// TIA Portal V19 export
TYPE "IF Burkett Type 8691 IO"
   STRUCT
      StandardStructure : Struct
         Header : Struct
            NumberParameter : Int := 56;   // Number of device parameters (Device Identification + Device Parameter)
            AdressParamDownLoad : Int := 20;   // Start adress for ParamDownload signals in this struct
            AdressDeviceIndent : Int := 44;   // Start adress for Device Identification Parameters in this struct
            AdressApplicSpez : Int := 700;   // Start adress ApplicationSpezificTag
            AdressDeviceParam : Int := 1110;   // Start adress for Device Parameters in this Area
            AdressKommando : Int := 1970;   // Start adress for Device Commandos
            NumberCommandos : Int := 4;   // Number of Commandos of the device
            Spare01 : Int;   // spare
            Spare02 : Int;   // spare
            Spare03 : Int;   // spare
         END_STRUCT;
         Paramdownload : Struct
            ParamDownLoadStart : Struct   // Parameter Download Start (Only if master and device are V1.1)
               BlockStat : DWord;   // function block status
               IOLStat : DWord;   // IO-Link Status
            END_STRUCT;
            ParamDownLoadEnd : Struct   // Parameter Download End (Only if master and device are V1.1)
               BlockStat : DWord;   // function block status
               IOLStat : DWord;   // IO-Link Status
            END_STRUCT;
            ParamDownLoadStore : Struct   // Parameter Download Store (Only if master and device are V1.1)
               BlockStat : DWord;   // function block status
               IOLStat : DWord;   // IO-Link Status
            END_STRUCT;
         END_STRUCT;
         DeviceIndentification : Struct   // device indentification parameter
            V_VendorName : Struct   // Vendor Name
               Text : String[64];
               Index : Int := 16;   // parameter index
               Subindex : Int;   // parameter subindex
               Length : Int := 64;   // parameter length in BYTE for writing
               BlockStat : DWord;   // function block status
               IOLStat : DWord;   // IO-Link Status
               RelRead : Bool := TRUE;   // reading release
               RelWrite : Bool;   // writing release
            END_STRUCT;
            V_VendorText : Struct   // Vendor Text
               Text : String[64];
               Index : Int := 17;   // parameter index
               Subindex : Int;   // parameter subindex
               Length : Int := 64;   // parameter length in BYTE for writing
               BlockStat : DWord;   // function block status
               IOLStat : DWord;   // IO-Link Status
               RelRead : Bool := TRUE;   // reading release
               RelWrite : Bool;   // writing release
            END_STRUCT;
            V_ProductName : Struct   // Product Name
               Text : String[64];
               Index : Int := 18;   // parameter index
               Subindex : Int;   // parameter subindex
               Length : Int := 64;   // parameter length in BYTE for writing
               BlockStat : DWord;   // function block status
               IOLStat : DWord;   // IO-Link Status
               RelRead : Bool := TRUE;   // reading release
               RelWrite : Bool;   // writing release
            END_STRUCT;
            V_ProductID : Struct   // Product ID
               Text : String[64];
               Index : Int := 19;   // parameter index
               Subindex : Int;   // parameter subindex
               Length : Int := 64;   // parameter length in BYTE for writing
               BlockStat : DWord;   // function block status
               IOLStat : DWord;   // IO-Link Status
               RelRead : Bool := TRUE;   // reading release
               RelWrite : Bool;   // writing release
            END_STRUCT;
            V_ProductText : Struct   // Product Text
               Text : String[64];
               Index : Int := 20;   // parameter index
               Subindex : Int;   // parameter subindex
               Length : Int := 64;   // parameter length in BYTE for writing
               BlockStat : DWord;   // function block status
               IOLStat : DWord;   // IO-Link Status
               RelRead : Bool := TRUE;   // reading release
               RelWrite : Bool;   // writing release
            END_STRUCT;
            V_SerialNumber : Struct   // Serial Number
               Text : String[64];
               Index : Int := 21;   // parameter index
               Subindex : Int;   // parameter subindex
               Length : Int := 16;   // parameter length in BYTE for writing
               BlockStat : DWord;   // function block status
               IOLStat : DWord;   // IO-Link Status
               RelRead : Bool := TRUE;   // reading release
               RelWrite : Bool;   // writing release
            END_STRUCT;
            V_HardwareRevision : Struct   // Hardware Version
               Text : String[64];
               Index : Int := 22;   // parameter index
               Subindex : Int;   // parameter subindex
               Length : Int := 64;   // parameter length in BYTE for writing
               BlockStat : DWord;   // function block status
               IOLStat : DWord;   // IO-Link Status
               RelRead : Bool := TRUE;   // reading release
               RelWrite : Bool;   // writing release
            END_STRUCT;
            V_FirmwareRevision : Struct   // Firmware Version
               Text : String[64];
               Index : Int := 23;   // parameter index
               Subindex : Int;   // parameter subindex
               Length : Int := 64;   // parameter length in BYTE for writing
               BlockStat : DWord;   // function block status
               IOLStat : DWord;   // IO-Link Status
               RelRead : Bool := TRUE;   // reading release
               RelWrite : Bool;   // writing release
            END_STRUCT;
         END_STRUCT;
         ApplicationSpecificTag : Struct   // AppliciationSpecificTag
            V_ApplicationSpecificTa : Struct   // Application Specific Tag
               Text : String[64];
               Index : Int := 24;   // parameter index
               Subindex : Int;   // parameter subindex
               Length : Int := 19;   // parameter length in BYTE for writing
               BlockStat : DWord;   // function block status
               IOLStat : DWord;   // IO-Link Status
               RelRead : Bool := TRUE;   // reading release
               RelWrite : Bool := TRUE;   // writing release
            END_STRUCT;
            V_UniqueDeviceName : Struct   // Name of Device
               Text : String[64];
               Index : Int := 8194;   // parameter index
               Subindex : Int := 1;   // parameter subindex
               Length : Int := 19;   // parameter length in BYTE for writing
               BlockStat : DWord;   // function block status
               IOLStat : DWord;   // IO-Link Status
               RelRead : Bool := TRUE;   // reading release
               RelWrite : Bool := TRUE;   // writing release
            END_STRUCT;
            V_LocationInformation : Struct   // Information about device location
               Text : String[64];
               Index : Int := 8194;   // parameter index
               Subindex : Int := 2;   // parameter subindex
               Length : Int := 19;   // parameter length in BYTE for writing
               BlockStat : DWord;   // function block status
               IOLStat : DWord;   // IO-Link Status
               RelRead : Bool := TRUE;   // reading release
               RelWrite : Bool := TRUE;   // writing release
            END_STRUCT;
            V_UserDescription : Struct   // Information about device
               Text : String[64];
               Index : Int := 8194;   // parameter index
               Subindex : Int := 3;   // parameter subindex
               Length : Int := 19;   // parameter length in BYTE for writing
               BlockStat : DWord;   // function block status
               IOLStat : DWord;   // IO-Link Status
               RelRead : Bool := TRUE;   // reading release
               RelWrite : Bool := TRUE;   // writing release
            END_STRUCT;
            V_DisplayedDeviceName : Struct   // Device (Tag) name
               Text : String[64];
               Index : Int := 8194;   // parameter index
               Subindex : Int := 4;   // parameter subindex
               Length : Int := 19;   // parameter length in BYTE for writing
               BlockStat : DWord;   // function block status
               IOLStat : DWord;   // IO-Link Status
               RelRead : Bool := TRUE;   // reading release
               RelWrite : Bool := TRUE;   // writing release
            END_STRUCT;
         END_STRUCT;
         DeviceParameters : Struct   // Device Parameters
            Parameter_00 : Struct
               Value : Struct   // Device Status
                  DeviceStatus : Byte;
                  byte_02 : Byte;
                  byte_03 : Byte;
                  byte_04 : Byte;
               END_STRUCT;
               Index : Int := 36;   // parameter index
               Subindex : Int;   // parameter subindex
               Length : Int := 1;   // parameter length in BYTE for writing
               BlockStat : DWord;   // function block status
               IOLStat : DWord;   // IO-Link Status
               RelRead : Bool := TRUE;   // reading release
               RelWrite : Bool;   // writing release
            END_STRUCT;
            Parameter_01 : Struct   // *** Control Head Settings - Index = 11276 ***
               Value : Struct   // Upper (open) tolerance band in mm
                  UTB : Real := 1.5;   // mm
               END_STRUCT;
               Index : Int := 11275;   // parameter index
               Subindex : Int := 1;   // parameter subindex
               Length : Int := 4;   // parameter length in BYTE for writing
               BlockStat : DWord;   // function block status
               IOLStat : DWord;   // IO-Link Status
               RelRead : Bool := TRUE;   // reading release
               RelWrite : Bool := TRUE;   // writing release
            END_STRUCT;
            Parameter_02 : Struct   // Control Head Settings - Lower (closed) tolerance band in mm
               Value : Struct   // Lower (closed) tolerance band in mm
                  LTB : Real := 1.5;   // mm Index = 11276
               END_STRUCT;
               Index : Int := 11275;   // parameter index
               Subindex : Int := 2;   // parameter subindex
               Length : Int := 4;   // parameter length in BYTE for writing
               BlockStat : DWord;   // function block status
               IOLStat : DWord;   // IO-Link Status
               RelRead : Bool := TRUE;   // reading release
               RelWrite : Bool := TRUE;   // writing release
            END_STRUCT;
            Parameter_03 : Struct   // Invert CMD Setpoint value
               Value : Struct   // Parameter Value (must be always 4 Byte)
                  InvertCMD_SP : Byte;   // 0=inversion inactive, 1=inversion inactive
                  Byte01 : Byte;
                  Byte02 : Byte;
                  Byte03 : Byte;
               END_STRUCT;
               Index : Int := 11275;   // parameter index
               Subindex : Int := 3;   // parameter subindex
               Length : Int := 1;   // parameter length in BYTE for writing
               BlockStat : DWord;   // function block status
               IOLStat : DWord;   // IO-Link Status
               RelRead : Bool := TRUE;   // reading release
               RelWrite : Bool := TRUE;   // writing release
            END_STRUCT;
            Parameter_04 : Struct   // Opening Time (CMD)
               Value : Struct   // Parameter Value (must be always 4 Byte)
                  OpeningTime : Int;   // ms
                  Byte02 : Byte;
                  Byte03 : Byte;
               END_STRUCT;
               Index : Int := 11275;   // parameter index
               Subindex : Int := 4;   // parameter subindex
               Length : Int := 2;   // parameter length in BYTE for writing
               BlockStat : DWord;   // function block status
               IOLStat : DWord;   // IO-Link Status
               RelRead : Bool := TRUE;   // reading release
               RelWrite : Bool;   // writing release
            END_STRUCT;
            Parameter_05 : Struct   // Closing Time (CMD)
               Value : Struct   // Parameter Value (must be always 4 Byte)
                  ClosingTime : Int;   // ms
                  Byte02 : Byte;
                  Byte03 : Byte;
               END_STRUCT;
               Index : Int := 11275;   // parameter index
               Subindex : Int := 5;   // parameter subindex
               Length : Int := 2;   // parameter length in BYTE for writing
               BlockStat : DWord;   // function block status
               IOLStat : DWord;   // IO-Link Status
               RelRead : Bool := TRUE;   // reading release
               RelWrite : Bool;   // writing release
            END_STRUCT;
            Parameter_06 : Struct   // Select reaction inevent of setpoint error
               Value : Struct   // Bus error or invalid process data
                  SetpointError : Byte;   // 0=Maintain position, 1=Safety position (pilot valve off)
                  Byte01 : Byte;
                  Byte02 : Byte;
                  Byte03 : Byte;
               END_STRUCT;
               Index : Int := 11275;   // parameter index
               Subindex : Int := 8;   // parameter subindex
               Length : Int := 1;   // parameter length in BYTE for writing
               BlockStat : DWord;   // function block status
               IOLStat : DWord;   // IO-Link Status
               RelRead : Bool := TRUE;   // reading release
               RelWrite : Bool := TRUE;   // writing release
            END_STRUCT;
            Parameter_07 : Struct   // Acitivate or deacitivate local operation
               Value : Struct   // Button for manula operation inside control head
                  DeviceLock : Byte;   // 0=Button enabled, 1=Button disabled
                  Byte01 : Byte;
                  Byte02 : Byte;
                  Byte03 : Byte;
               END_STRUCT;
               Index : Int := 11275;   // parameter index
               Subindex : Int := 12;   // parameter subindex
               Length : Int := 1;   // parameter length in BYTE for writing
               BlockStat : DWord;   // function block status
               IOLStat : DWord;   // IO-Link Status
               RelRead : Bool := TRUE;   // reading release
               RelWrite : Bool := TRUE;   // writing release
            END_STRUCT;
            Parameter_08 : Struct   // *** Teach Functions Index = 11276 ***
               Value : Struct   // Parameter Value (must be always 4 Byte)
                  UpperEndPosition : Real;
               END_STRUCT;
               Index : Int := 11276;   // parameter index
               Subindex : Int := 1;   // parameter subindex
               Length : Int := 4;   // parameter length in BYTE for writing
               BlockStat : DWord;   // function block status
               IOLStat : DWord;   // IO-Link Status
               RelRead : Bool := TRUE;   // reading release
               RelWrite : Bool;   // writing release
            END_STRUCT;
            Parameter_09 : Struct   // *** Teach Functions Index = 11276 ***
               Value : Struct   // Parameter Value (must be always 4 Byte)
                  LowerEndPosition : Real;
               END_STRUCT;
               Index : Int := 11276;   // parameter index
               Subindex : Int := 2;   // parameter subindex
               Length : Int := 4;   // parameter length in BYTE for writing
               BlockStat : DWord;   // function block status
               IOLStat : DWord;   // IO-Link Status
               RelRead : Bool := TRUE;   // reading release
               RelWrite : Bool;   // writing release
            END_STRUCT;
            Parameter_10 : Struct   // *** Teach Functions Index = 11276 ***
               Value : Struct   // Opening Time between tolerance bands
                  Opening_Time : Int;   // ms
                  Byte02 : Byte;
                  Byte03 : Byte;
               END_STRUCT;
               Index : Int := 11276;   // parameter index
               Subindex : Int := 3;   // parameter subindex
               Length : Int := 2;   // parameter length in BYTE for writing
               BlockStat : DWord;   // function block status
               IOLStat : DWord;   // IO-Link Status
               RelRead : Bool := TRUE;   // reading release
               RelWrite : Bool;   // writing release
            END_STRUCT;
            Parameter_11 : Struct   // *** Teach Functions Index = 11276 ***
               Value : Struct   // Closing Time between tolerance bands
                  Closing_Time : Int;   // ms
                  Byte02 : Byte;
                  Byte03 : Byte;
               END_STRUCT;
               Index : Int := 11276;   // parameter index
               Subindex : Int := 4;   // parameter subindex
               Length : Int := 2;   // parameter length in BYTE for writing
               BlockStat : DWord;   // function block status
               IOLStat : DWord;   // IO-Link Status
               RelRead : Bool := TRUE;   // reading release
               RelWrite : Bool;   // writing release
            END_STRUCT;
            Parameter_12 : Struct   // *** Teach Functions Index = 11276 ***
               Value : Struct   // Parameter Value (must be always 4 Byte)
                  Stroke : Real;   // Valve stroke in mm
               END_STRUCT;
               Index : Int := 11276;   // parameter index
               Subindex : Int := 5;   // parameter subindex
               Length : Int := 4;   // parameter length in BYTE for writing
               BlockStat : DWord;   // function block status
               IOLStat : DWord;   // IO-Link Status
               RelRead : Bool := TRUE;   // reading release
               RelWrite : Bool;   // writing release
            END_STRUCT;
            Parameter_14 : Struct   // Is Teached
               Value : Struct   // Indicates successful completion of a teach funtion
                  IsTeached : Byte;   // 0=Device has not been taught, 1=Device taught
                  Byte01 : Byte;
                  Byte02 : Byte;
                  Byte03 : Byte;
               END_STRUCT;
               Index : Int := 11276;   // parameter index
               Subindex : Int := 6;   // parameter subindex
               Length : Int := 1;   // parameter length in BYTE for writing
               BlockStat : DWord;   // function block status
               IOLStat : DWord;   // IO-Link Status
               RelRead : Bool := TRUE;   // reading release
               RelWrite : Bool;   // writing release
            END_STRUCT;
            Parameter_15 : Struct   // Teach function State
               Value : Struct   // 0=complete,1=Initialisation,2=End Position1,3=End Position2,4=Check Stroke,
                  TeachFuncState : Byte;   // 5=DetermineSwitchingTime,-1=TimeoutEndPos1,-2=TimeoutEndPos2
                  Byte01 : Byte;   // -3=StrokeTooSmall,-4=ErrorDeterminingSwitchingTime,
                  Byte02 : Byte;   // -5=AbortbySafePos, -6=AbortbyUser
                  Byte03 : Byte;
               END_STRUCT;
               Index : Int := 11276;   // parameter index
               Subindex : Int := 7;   // parameter subindex
               Length : Int := 1;   // parameter length in BYTE for writing
               BlockStat : DWord;   // function block status
               IOLStat : DWord;   // IO-Link Status
               RelRead : Bool := TRUE;   // reading release
               RelWrite : Bool;   // writing release
            END_STRUCT;
            Parameter_16 : Struct   // Start Teach function
               Value : Struct
                  TeachFuncStart : Byte;   // 0 = Finished,1 = StartAutomaticTeach, 2 = StartManualTeach
                  Byte01 : Byte;
                  Byte02 : Byte;
                  Byte03 : Byte;
               END_STRUCT;
               Index : Int := 11276;   // parameter index
               Subindex : Int := 8;   // parameter subindex
               Length : Int := 1;   // parameter length in BYTE for writing
               BlockStat : DWord;   // function block status
               IOLStat : DWord;   // IO-Link Status
               RelRead : Bool := TRUE;   // reading release
               RelWrite : Bool := TRUE;   // writing release
            END_STRUCT;
            Parameter_17 : Struct   // Flag shows pneumatic function
               Value : Struct
                  isNO : Byte;   // 0 = Normally Closed (NC), 1 = Normally Open (NO)
                  Byte01 : Byte;
                  Byte02 : Byte;
                  Byte03 : Byte;
               END_STRUCT;
               Index : Int := 11276;   // parameter index
               Subindex : Int := 9;   // parameter subindex
               Length : Int := 1;   // parameter length in BYTE for writing
               BlockStat : DWord;   // function block status
               IOLStat : DWord;   // IO-Link Status
               RelRead : Bool := TRUE;   // reading release
               RelWrite : Bool;   // writing release
            END_STRUCT;
            Parameter_18 : Struct   // Select CMD set-point value source
               Value : Struct
                  CMD_Source : Byte := BYTE#16#01;   // 1 = IO-Link (Cyclic or via SIO),2 = InternalButton, 3 = ManualSPValue(sub0x4)
                  Byte01 : Byte;
                  Byte02 : Byte;
                  Byte03 : Byte;
               END_STRUCT;
               Index : Int := 11277;   // parameter index
               Subindex : Int := 1;   // parameter subindex
               Length : Int := 1;   // parameter length in BYTE for writing
               BlockStat : DWord;   // function block status
               IOLStat : DWord;   // IO-Link Status
               RelRead : Bool := TRUE;   // reading release
               RelWrite : Bool := TRUE;   // writing release
            END_STRUCT;
            Parameter_19 : Struct   // Manual CMD Set-point
               Value : Struct
                  Manual_CMD_SP : Byte;
                  Byte01 : Byte;
                  Byte02 : Byte;
                  Byte03 : Byte;
               END_STRUCT;
               Index : Int := 11277;   // parameter index
               Subindex : Int := 4;   // parameter subindex
               Length : Int := 1;   // parameter length in BYTE for writing
               BlockStat : DWord;   // function block status
               IOLStat : DWord;   // IO-Link Status
               RelRead : Bool := TRUE;   // reading release
               RelWrite : Bool := TRUE;   // writing release
            END_STRUCT;
            Parameter_20 : Struct   // *** Diagnostics , Index = 11278 ***
               Value : Struct
                  TravelAccumlator : Real;   // Valve stem travel in mm
               END_STRUCT;
               Index : Int := 11278;   // parameter index
               Subindex : Int := 1;   // parameter subindex
               Length : Int := 4;   // parameter length in BYTE for writing
               BlockStat : DWord;   // function block status
               IOLStat : DWord;   // IO-Link Status
               RelRead : Bool := TRUE;   // reading release
               RelWrite : Bool;   // writing release
            END_STRUCT;
            Parameter_21 : Struct   // *** Diagnostics , Index = 11278 ***
               Value : Struct
                  TravelAccResettable : Real;   // Valve stem travel in mm
               END_STRUCT;
               Index : Int := 11278;   // parameter index
               Subindex : Int := 2;   // parameter subindex
               Length : Int := 4;   // parameter length in BYTE for writing
               BlockStat : DWord;   // function block status
               IOLStat : DWord;   // IO-Link Status
               RelRead : Bool := TRUE;   // reading release
               RelWrite : Bool;   // writing release
            END_STRUCT;
            Parameter_22 : Struct   // Travel Accumulator in mm, Activate or deactivate maintenance threshold
               Value : Struct
                  TravelAccLimit : Real;   // Travel Acc Limit in mm
               END_STRUCT;
               Index : Int := 11278;   // parameter index
               Subindex : Int := 3;   // parameter subindex
               Length : Int := 4;   // parameter length in BYTE for writing
               BlockStat : DWord;   // function block status
               IOLStat : DWord;   // IO-Link Status
               RelRead : Bool := TRUE;   // reading release
               RelWrite : Bool := TRUE;   // writing release
            END_STRUCT;
            Parameter_23 : Struct   // Valve Cycles
               Value : Struct
                  ValveCycles : DInt;   // # of Valve Cycles
               END_STRUCT;
               Index : Int := 11278;   // parameter index
               Subindex : Int := 4;   // parameter subindex
               Length : Int := 4;   // parameter length in BYTE for writing
               BlockStat : DWord;   // function block status
               IOLStat : DWord;   // IO-Link Status
               RelRead : Bool := TRUE;   // reading release
               RelWrite : Bool;   // writing release
            END_STRUCT;
            Parameter_24 : Struct   // Valve Cycles Resetable
               Value : Struct
                  ValveCyclesResettable : DInt;   // # of Valve Cycles
               END_STRUCT;
               Index : Int := 11278;   // parameter index
               Subindex : Int := 5;   // parameter subindex
               Length : Int := 4;   // parameter length in BYTE for writing
               BlockStat : DWord;   // function block status
               IOLStat : DWord;   // IO-Link Status
               RelRead : Bool := TRUE;   // reading release
               RelWrite : Bool;   // writing release
            END_STRUCT;
            Parameter_25 : Struct   // Valve Cycles Limit
               Value : Struct   // ValveCyclesResetable > ValveCyclesLimit = Activate Maintenance Warning
                  ValveCyclesLimit : DInt;   // # of Valve Cycles
               END_STRUCT;
               Index : Int := 11278;   // parameter index
               Subindex : Int := 6;   // parameter subindex
               Length : Int := 4;   // parameter length in BYTE for writing
               BlockStat : DWord;   // function block status
               IOLStat : DWord;   // IO-Link Status
               RelRead : Bool := TRUE;   // reading release
               RelWrite : Bool := TRUE;   // writing release
            END_STRUCT;
            Parameter_26 : Struct   // Operating Time Resettable
               Value : Struct   // Sum of time device recieving operating voltage
                  OperateTimeResettable : DInt;   // time in seconds
               END_STRUCT;
               Index : Int := 11278;   // parameter index
               Subindex : Int := 7;   // parameter subindex
               Length : Int := 4;   // parameter length in BYTE for writing
               BlockStat : DWord;   // function block status
               IOLStat : DWord;   // IO-Link Status
               RelRead : Bool := TRUE;   // reading release
               RelWrite : Bool;   // writing release
            END_STRUCT;
            Parameter_27 : Struct   // Operating Time Limit
               Value : Struct   // OperateTimeResetable > OperateTimeLimit = Activate Maintenance Warning
                  OperateTimeLimit : DInt;   // time in seconds
               END_STRUCT;
               Index : Int := 11278;   // parameter index
               Subindex : Int := 8;   // parameter subindex
               Length : Int := 4;   // parameter length in BYTE for writing
               BlockStat : DWord;   // function block status
               IOLStat : DWord;   // IO-Link Status
               RelRead : Bool := TRUE;   // reading release
               RelWrite : Bool := TRUE;   // writing release
            END_STRUCT;
            Parameter_28 : Struct   // Diagnostics Command
               Value : Struct   // Bit0=ResetSwitchingCycles, Bit1=ResetTravelACC, Bit2=ResetOperateTime
                  Diag_CMD : Byte;   // Bit3=Reset#OfOpeningTimeTimeouts,Bit4=Reset#OfClosingTimeTimeouts,
                  Byte01 : Byte;   // Bit5=CopyMeasuredSwitchingTimes, Bit6=ResetNoOfSwitchingTimeTimeouts
                  Byte02 : Byte;
                  Byte03 : Byte;
               END_STRUCT;
               Index : Int := 11278;   // parameter index
               Subindex : Int := 9;   // parameter subindex
               Length : Int := 1;   // parameter length in BYTE for writing
               BlockStat : DWord;   // function block status
               IOLStat : DWord;   // IO-Link Status
               RelRead : Bool := TRUE;   // reading release
               RelWrite : Bool := TRUE;   // writing release
            END_STRUCT;
            Parameter_29 : Struct   // ** Maximum Opening Time in ms **
               Value : Struct
                  OpeningTimeLimit : Int;   // ms
                  Byte02 : Byte;
                  Byte03 : Byte;
               END_STRUCT;
               Index : Int := 11278;   // parameter index
               Subindex : Int := 10;   // parameter subindex
               Length : Int := 2;   // parameter length in BYTE for writing
               BlockStat : DWord;   // function block status
               IOLStat : DWord;   // IO-Link Status
               RelRead : Bool := TRUE;   // reading release
               RelWrite : Bool := TRUE;   // writing release
            END_STRUCT;
            Parameter_30 : Struct   // ** Maximum Closing Time in ms **
               Value : Struct
                  ClosingTimeLimit : Int;   // ms
                  Byte02 : Byte;
                  Byte03 : Byte;
               END_STRUCT;
               Index : Int := 11278;   // parameter index
               Subindex : Int := 11;   // parameter subindex
               Length : Int := 2;   // parameter length in BYTE for writing
               BlockStat : DWord;   // function block status
               IOLStat : DWord;   // IO-Link Status
               RelRead : Bool := TRUE;   // reading release
               RelWrite : Bool := TRUE;   // writing release
            END_STRUCT;
            Parameter_31 : Struct   // Time Tolerance
               Value : Struct
                  TimeTolerance : Byte;   // %
                  Byte01 : Byte;
                  Byte02 : Byte;
                  Byte03 : Byte;
               END_STRUCT;
               Index : Int := 11278;   // parameter index
               Subindex : Int := 12;   // parameter subindex
               Length : Int := 1;   // parameter length in BYTE for writing
               BlockStat : DWord;   // function block status
               IOLStat : DWord;   // IO-Link Status
               RelRead : Bool := TRUE;   // reading release
               RelWrite : Bool := TRUE;   // writing release
            END_STRUCT;
            Parameter_32 : Struct   // Opening Time Errors
               Value : Struct
                  OpeningTimeErrors : DInt;   // # of Opening Time Errors - Resettable
               END_STRUCT;
               Index : Int := 11278;   // parameter index
               Subindex : Int := 13;   // parameter subindex
               Length : Int := 4;   // parameter length in BYTE for writing
               BlockStat : DWord;   // function block status
               IOLStat : DWord;   // IO-Link Status
               RelRead : Bool := TRUE;   // reading release
               RelWrite : Bool;   // writing release
            END_STRUCT;
            Parameter_33 : Struct   // Closing Time Errors
               Value : Struct
                  ClosingTimeErrors : DInt;   // # of Closing Time Errors - Resettable
               END_STRUCT;
               Index : Int := 11278;   // parameter index
               Subindex : Int := 14;   // parameter subindex
               Length : Int := 4;   // parameter length in BYTE for writing
               BlockStat : DWord;   // function block status
               IOLStat : DWord;   // IO-Link Status
               RelRead : Bool := TRUE;   // reading release
               RelWrite : Bool;   // writing release
            END_STRUCT;
            Parameter_34 : Struct   // Teach Function Counter
               Value : Struct
                  TeachFuncCounter : DInt;   // # of Teach Functions Preformed
               END_STRUCT;
               Index : Int := 11278;   // parameter index
               Subindex : Int := 15;   // parameter subindex
               Length : Int := 4;   // parameter length in BYTE for writing
               BlockStat : DWord;   // function block status
               IOLStat : DWord;   // IO-Link Status
               RelRead : Bool := TRUE;   // reading release
               RelWrite : Bool;   // writing release
            END_STRUCT;
            Parameter_35 : Struct   // Pilot Valve Cycles Counter
               Value : Struct
                  PilotValveCycles : DInt;   // # of Pilot Valve Cycles
               END_STRUCT;
               Index : Int := 11278;   // parameter index
               Subindex : Int := 16;   // parameter subindex
               Length : Int := 4;   // parameter length in BYTE for writing
               BlockStat : DWord;   // function block status
               IOLStat : DWord;   // IO-Link Status
               RelRead : Bool := TRUE;   // reading release
               RelWrite : Bool;   // writing release
            END_STRUCT;
            Parameter_36 : Struct   // Number of Switching Timeouts
               Value : Struct
                  SwitchingTimeouts : DInt;   // # of Switching Timeouts
               END_STRUCT;
               Index : Int := 11278;   // parameter index
               Subindex : Int := 18;   // parameter subindex
               Length : Int := 4;   // parameter length in BYTE for writing
               BlockStat : DWord;   // function block status
               IOLStat : DWord;   // IO-Link Status
               RelRead : Bool := TRUE;   // reading release
               RelWrite : Bool;   // writing release
            END_STRUCT;
            Parameter_37 : Struct   // Select type of switching times for diagnostics
               Value : Struct
                  TimeDiagType : Byte;   // 0=Switching Time Based on CMD, 1=Switching Time Based on position
                  Byte01 : Byte;
                  Byte02 : Byte;
                  Byte03 : Byte;
               END_STRUCT;
               Index : Int := 11278;   // parameter index
               Subindex : Int := 21;   // parameter subindex
               Length : Int := 1;   // parameter length in BYTE for writing
               BlockStat : DWord;   // function block status
               IOLStat : DWord;   // IO-Link Status
               RelRead : Bool := TRUE;   // reading release
               RelWrite : Bool := TRUE;   // writing release
            END_STRUCT;
            Parameter_38 : Struct   // Activate or deactivate switching time timeout detection.
               Value : Struct
                  SwitchingTimeoutDetect : Byte := BYTE#16#01;   // 0=Deactivated, 1=Activated
                  Byte01 : Byte;
                  Byte02 : Byte;
                  Byte03 : Byte;
               END_STRUCT;
               Index : Int := 11278;   // parameter index
               Subindex : Int := 23;   // parameter subindex
               Length : Int := 1;   // parameter length in BYTE for writing
               BlockStat : DWord;   // function block status
               IOLStat : DWord;   // IO-Link Status
               RelRead : Bool := TRUE;   // reading release
               RelWrite : Bool := TRUE;   // writing release
            END_STRUCT;
            Parameter_39 : Struct   // Select max time in ms by which the end position should be reached
               Value : Struct
                  SwitchingTimeout : Int := 500;   // ms
                  Byte02 : Byte;
                  Byte03 : Byte;
               END_STRUCT;
               Index : Int := 11278;   // parameter index
               Subindex : Int := 24;   // parameter subindex
               Length : Int := 2;   // parameter length in BYTE for writing
               BlockStat : DWord;   // function block status
               IOLStat : DWord;   // IO-Link Status
               RelRead : Bool := TRUE;   // reading release
               RelWrite : Bool := TRUE;   // writing release
            END_STRUCT;
            Parameter_40 : Struct   // SIO Mode
               Value : Struct   // Pin 2 / Pin 4
                  SIO_Mode : Byte;   // 0=Open/Close, 1=CMD/Close, 2=CMD/Open
                  Byte01 : Byte;   // ** DEVICE MUST BE RESTARTED IF VALUE CHANGED **
                  Byte02 : Byte;
                  Byte03 : Byte;
               END_STRUCT;
               Index : Int := 11279;   // parameter index
               Subindex : Int := 1;   // parameter subindex
               Length : Int := 1;   // parameter length in BYTE for writing
               BlockStat : DWord;   // function block status
               IOLStat : DWord;   // IO-Link Status
               RelRead : Bool := TRUE;   // reading release
               RelWrite : Bool := TRUE;   // writing release
            END_STRUCT;
            Parameter_41 : Struct   // Output Type
               Value : Struct
                  OutputType : Byte;   // 0=PNP, 1=NPN, 2=PP
                  Byte01 : Byte;   // ** DEVICE MUST BE RESTARTED IF VALUE CHANGED **
                  Byte02 : Byte;
                  Byte03 : Byte;
               END_STRUCT;
               Index : Int := 11279;   // parameter index
               Subindex : Int := 1;   // parameter subindex
               Length : Int := 1;   // parameter length in BYTE for writing
               BlockStat : DWord;   // function block status
               IOLStat : DWord;   // IO-Link Status
               RelRead : Bool := TRUE;   // reading release
               RelWrite : Bool := TRUE;   // writing release
            END_STRUCT;
            Parameter_42 : Struct   // Invert Valve Direction
               Value : Struct
                  InvValveDir : Byte;   // 0=UpperPos/Open, 1=UpperPos/Closed
                  Byte01 : Byte;
                  Byte02 : Byte;
                  Byte03 : Byte;
               END_STRUCT;
               Index : Int := 11268;   // parameter index
               Subindex : Int := 1;   // parameter subindex
               Length : Int := 1;   // parameter length in BYTE for writing
               BlockStat : DWord;   // function block status
               IOLStat : DWord;   // IO-Link Status
               RelRead : Bool := TRUE;   // reading release
               RelWrite : Bool := TRUE;   // writing release
            END_STRUCT;
            Parameter_43 : Struct   // CMD Setpoint Control Mode
               Value : Struct
                  CMD_SP_CNTRL_MODE : Byte;
                  Byte01 : Byte;
                  Byte02 : Byte;
                  Byte03 : Byte;
               END_STRUCT;
               Index : Int := 11268;   // parameter index
               Subindex : Int := 2;   // parameter subindex
               Length : Int := 1;   // parameter length in BYTE for writing
               BlockStat : DWord;   // function block status
               IOLStat : DWord;   // IO-Link Status
               RelRead : Bool := TRUE;   // reading release
               RelWrite : Bool := TRUE;   // writing release
            END_STRUCT;
         END_STRUCT;
         Commando : Struct   // Commandos
            Commando_01 : Struct   // Device Reset
               Value : Byte := BYTE#16#80;   // 128
               Index : Int := 2;   // parameter index
               Subindex : Int;   // parameter subindex
               Length : Int := 1;   // parameter length in BYTE for writing
               BlockStat : DWord;   // function block status
               IOLStat : DWord;   // IO-Link Status
            END_STRUCT;
            Commando_02 : Struct   // Restroe factory settings
               Value : Byte := BYTE#16#28;   // 130
               Index : Int := 2;   // parameter index
               Subindex : Int;   // parameter subindex
               Length : Int := 1;   // parameter length in BYTE for writing
               BlockStat : DWord;   // function block status
               IOLStat : DWord;   // IO-Link Status
            END_STRUCT;
            Commando_03 : Struct   // Start automatic Teach-function
               Value : Byte := BYTE#16#A0;   // 160
               Index : Int := 2;   // parameter index
               Subindex : Int;   // parameter subindex
               Length : Int := 1;   // parameter length in BYTE for writing
               BlockStat : DWord;   // function block status
               IOLStat : DWord;   // IO-Link Status
            END_STRUCT;
            Commando_04 : Struct   // Start manual Teach-function
               Value : Byte := BYTE#16#A1;
               Index : Int := 2;   // parameter index
               Subindex : Int;   // parameter subindex
               Length : Int := 1;   // parameter length in BYTE for writing
               BlockStat : DWord;   // function block status
               IOLStat : DWord;   // IO-Link Status
            END_STRUCT;
         END_STRUCT;
      END_STRUCT;
   END_STRUCT;
END_TYPE
